// TwinCAT 3 PLC project Untitled1
// ProgramVersion: 3.1.4023.0
// libraries:
//   Tc2_Standard, * (Beckhoff Automation GmbH)
//   Tc2_System, * (Beckhoff Automation GmbH)
//   Tc3_Module, * (Beckhoff Automation GmbH)
// project tree:
//   DUTs/ T_person.TcDUT
//   POUs/ BirthdayManager.TcPOU, BirthdayManager_1.TcPOU, MAIN.TcPOU
//   / Task_2.TcTTO
// real-time tasks:
//   TASK Task 2: cycle T#1ms, priority 1, ADS port 301
// I/O:
//   DEVICE Device 2 (CX-BK) (disabled)
//     Box 1 (CX-BK)
// variable links:
//   Untitled1/Untitled1 Instance <-> Device 2 (CX-BK)/Box 1 (CX-BK)
//     Task_2 Inputs/MAIN.potentioneter1 <-> Term 4 (KL3464)/Channel 1/Data In
//     Task_2 Inputs/MAIN.switch3 <-> Term 2 (KL1408)/Channel 2/Input
//     Task_2 Inputs/MAIN.switch4 <-> Term 2 (KL1408)/Channel 4/Input
//     Task_2 Inputs/MAIN.switches[{0..3}] <-> Term 2 (KL1408)/Channel {5..8}/Input  (4 links)
//     Task_2 Outputs/MAIN.Voltage <-> Term 5 (KL4002)/Channel 1/Data Out
//   Task 2 <-> Device 2 (CX-BK)/Box 1 (CX-BK)
//     Inputs/Switch 1 <-> Term 2 (KL1408)/Channel 1/Input
//     Inputs/Switch 2 <-> Term 2 (KL1408)/Channel 3/Input

CONFIGURATION Untitled1
    RESOURCE PLC ON TwinCAT3
        TASK Task_2(INTERVAL := T#10ms, PRIORITY := 1);
        PROGRAM MAIN WITH Task_2 : MAIN;
    END_RESOURCE
END_CONFIGURATION

// ---- DUTs/T_person.TcDUT
TYPE T_person :
STRUCT
	name:	STRING;
	age:	USINT;
	birthday: DATE;
END_STRUCT
END_TYPE

// ---- POUs/MAIN.TcPOU
PROGRAM MAIN
VAR
	
	counter: UINT := 0;
	switch3 AT%I*:BOOL;
	switch4 AT%I*:BOOL;
	Voltage AT%Q*:UINT;
	Voltage1 AT%Q*:UINT;
	switches AT%I*:ARRAY[0..3]OF	BOOL;
	potentioneter1 AT%I*:INT;
	fbBM: BirthdayManager_1;
END_VAR

counter:=counter+1;
voltage1:=potentioneter1;
FOR counter:=1 TO 1000 DO
	;
END_FOR


fbBM();

END_PROGRAM

// ---- POUs/BirthdayManager_1.TcPOU
FUNCTION_BLOCK BirthdayManager_1
VAR
	current_date:DATE:=D#2021-7-27;
	person:ARRAY[1..10]OF	T_person:=[(name:='Ali',age:=30,birthday:=D#2020-7-27),
										(name:='Ali',age:=30,birthday:=D#2020-7-27),
										(name:='Ali',age:=30,birthday:=D#2020-7-27),
										(name:='Azmi',age:=36,birthday:=D#2021-7-27),
										(name:='Ali',age:=30,birthday:=D#2020-7-27)];
	i: INT;
	message:string;
	execute: BOOL;
END_VAR

IF	execute	THEN
	FOR i:=1	TO	10	DO
		IF	person[i].birthday=current_date	THEN
			message:='happy Birthday ';
			message:=CONCAT(message,person[i].name);
			person[i].age:=person[i].age+1;
			message:=concat(message,' you are now ');
			message:=concat(message,USINT_TO_STRING(person[i].age));
			execute:=FALSE;
			RETURN;
		END_IF
	END_FOR
END_IF

END_FUNCTION_BLOCK

// ---- POUs/BirthdayManager.TcPOU
FUNCTION_BLOCK BirthdayManager
VAR
	current_date:DATE:=D#2021-7-27;
	names:ARRAY[1..10]OF	STRING:=['Ali','Azmi','Usama','Arsham'];
	age:ARRAY[1..10]OF	USINT(0..125):=[10,10,10,35];
	birthday:ARRAY[1..10]OF DATE:=[D#2020-7-27,D#2020-7-27,D#2020-7-27,D#2021-7-27];
	i: INT;
	message:string;
	execute: BOOL;
END_VAR

IF	execute	THEN
	FOR i:=1	TO	10	DO
		IF	birthday[i]=current_date	THEN
			message:='happy Birthday ';
			message:=CONCAT(message,names[i]);
			age[i]:=age[i]+1;
			message:=concat(message,' you are now ');
			message:=concat(message,USINT_TO_STRING(age[i]));
			execute:=FALSE;
			RETURN;
		END_IF
	END_FOR
END_IF

END_FUNCTION_BLOCK
